// TIA Portal V17 export
// export: Created 2023-09-10T16:27:48.4257814Z, ExportSetting WithDefaults, DisplayName Totally Integrated Automation Portal, DisplayVersion V17, DisplayName TIA Portal Openness, DisplayVersion V17, DisplayName TIA Portal Version Control Interface, DisplayVersion V17, DisplayName STEP 7 Professional, DisplayVersion V17, DisplayName STEP 7 Safety, DisplayVersion V17, DisplayName WinCC Advanced, DisplayVersion V17
ORGANIZATION_BLOCK "Main"   // OB1, LAD, ProgramCycle
TITLE = "Main Program Sweep (Cycle)"
{ S7_Optimized_Access := 'TRUE' }
VERSION : 0.1
// stored: AutoNumber true, IsIECCheckEnabled false, SetENOAutomatically false
   VAR_INPUT
      Initial_Call : Bool;   // Initial call of this OB
      Remanence : Bool;   // =True, if remanent data are available
   END_VAR
   VAR_TEMP
      turn : Int;
      machinePosition : DInt;
   END_VAR
   VAR_TEMP   // added for the SCL form of the ladder/FBD networks
      _w1 : Bool;
      _w2 : Bool;
      _w3 : Bool;
   END_VAR
BEGIN

REGION Network 1: Encoder modbus function
   // te
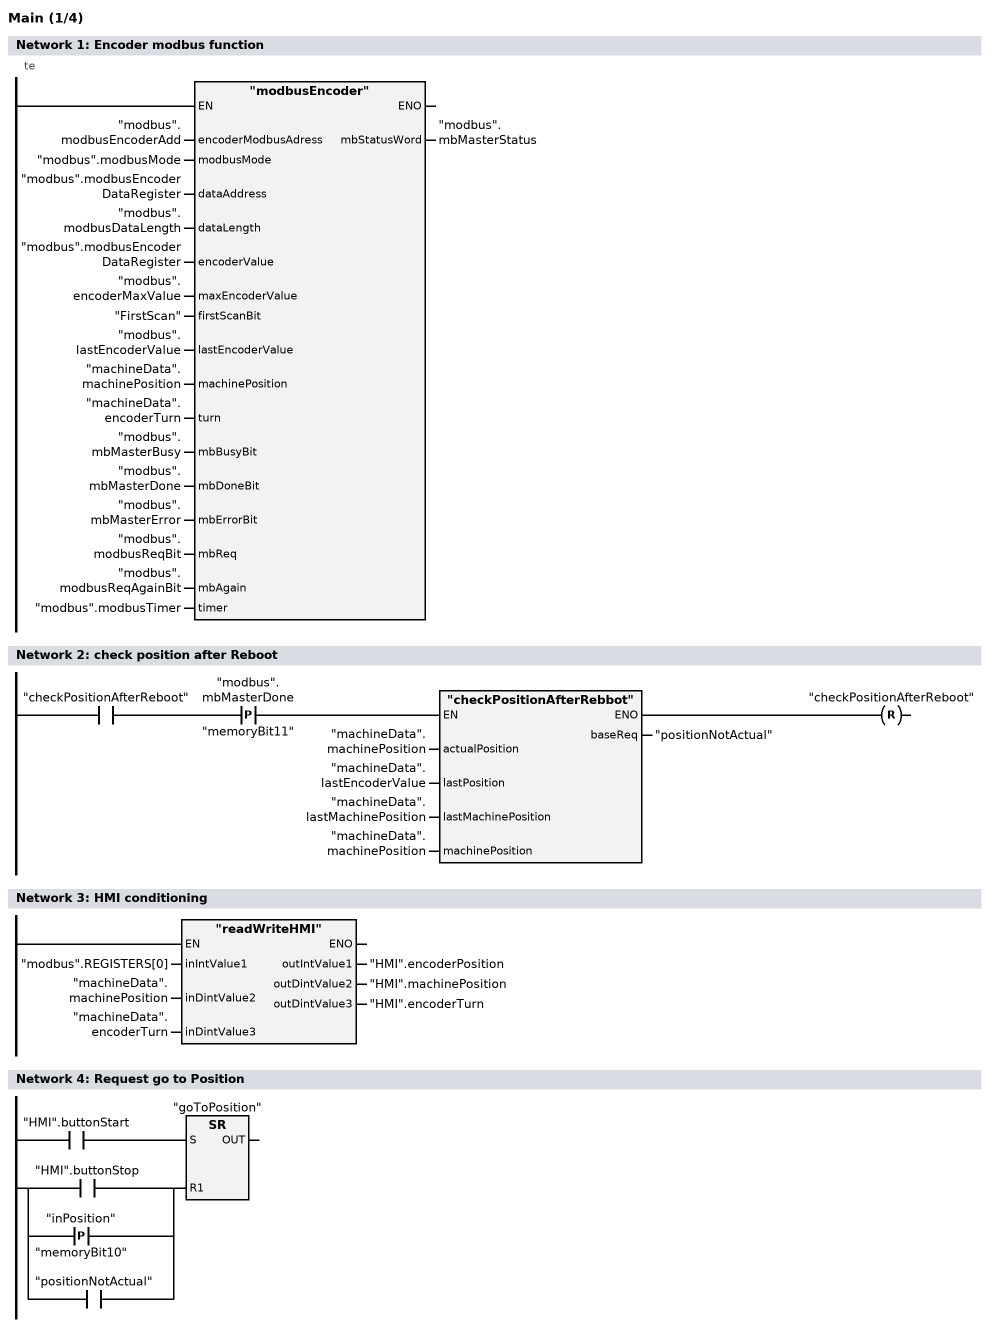
   RUNG wire#powerrail
      "modbusEncoder"(encoderModbusAdress := "modbus".modbusEncoderAdd, modbusMode := "modbus".modbusMode, dataAddress := "modbus".modbusEncoderDataRegister, dataLength := "modbus".modbusDataLength, encoderValue := "modbus".modbusEncoderDataRegister, maxEncoderValue := "modbus".encoderMaxValue, firstScanBit := "FirstScan", lastEncoderValue := "modbus".lastEncoderValue, machinePosition := "machineData".machinePosition, turn := "machineData".encoderTurn, mbBusyBit := "modbus".mbMasterBusy, mbDoneBit := "modbus".mbMasterDone, mbErrorBit := "modbus".mbMasterError, mbReq := "modbus".modbusReqBit, mbAgain := "modbus".modbusReqAgainBit, "timer" := "modbus".modbusTimer, mbStatusWord => "modbus".mbMasterStatus)
   END_RUNG
   // the same network as SCL:
   "modbusEncoder"(encoderModbusAdress := "modbus".modbusEncoderAdd,
                   modbusMode := "modbus".modbusMode,
                   dataAddress := "modbus".modbusEncoderDataRegister,
                   dataLength := "modbus".modbusDataLength,
                   encoderValue := "modbus".modbusEncoderDataRegister,
                   maxEncoderValue := "modbus".encoderMaxValue,
                   firstScanBit := "FirstScan",
                   lastEncoderValue := "modbus".lastEncoderValue,
                   machinePosition := "machineData".machinePosition,
                   turn := "machineData".encoderTurn,
                   mbBusyBit := "modbus".mbMasterBusy,
                   mbDoneBit := "modbus".mbMasterDone,
                   mbErrorBit := "modbus".mbMasterError,
                   mbReq := "modbus".modbusReqBit,
                   mbAgain := "modbus".modbusReqAgainBit,
                   "timer" := "modbus".modbusTimer,
                   mbStatusWord => "modbus".mbMasterStatus);
END_REGION

REGION Network 2: check position after Reboot
   RUNG wire#powerrail
      Contact( "checkPositionAfterReboot" )
      P_Contact(operand := "modbus".mbMasterDone, bit := "memoryBit11")
      "checkPositionAfterRebbot"(actualPosition := "machineData".machinePosition, lastPosition := "machineData".lastEncoderValue, lastMachinePosition := "machineData".lastMachinePosition, machinePosition := "machineData".machinePosition, baseReq => "positionNotActual")
      R_Coil( "checkPositionAfterReboot" )
   END_RUNG
   // the same network as SCL:
   #_w1 := "checkPositionAfterReboot" AND "modbus".mbMasterDone AND NOT "memoryBit11";   // rising edge of "modbus".mbMasterDone
   "memoryBit11" := "modbus".mbMasterDone;
   "checkPositionAfterRebbot"(EN := #_w1,
                           actualPosition := "machineData".machinePosition,
                           lastPosition := "machineData".lastEncoderValue,
                           lastMachinePosition := "machineData".lastMachinePosition,
                           machinePosition := "machineData".machinePosition,
                           baseReq => "positionNotActual",
                           ENO => #_w2);
   IF #_w2 THEN "checkPositionAfterReboot" := FALSE; END_IF;
END_REGION

REGION Network 3: HMI conditioning
   RUNG wire#powerrail
      "readWriteHMI"(inIntValue1 := "modbus".REGISTERS[0], inDintValue2 := "machineData".machinePosition, inDintValue3 := "machineData".encoderTurn, outIntValue1 => "HMI".encoderPosition, outDintValue2 => "HMI".machinePosition, outDintValue3 => "HMI".encoderTurn)
   END_RUNG
   // the same network as SCL:
   "readWriteHMI"(inIntValue1 := "modbus".REGISTERS[0],
                  inDintValue2 := "machineData".machinePosition,
                  inDintValue3 := "machineData".encoderTurn,
                  outIntValue1 => "HMI".encoderPosition,
                  outDintValue2 => "HMI".machinePosition,
                  outDintValue3 => "HMI".encoderTurn);
END_REGION

REGION Network 4: Request go to Position
   RUNG wire#powerrail
      Contact( "HMI".buttonStart )
      S_SR(operand := "goToPosition", r1 := wire#w1)
   END_RUNG
   RUNG wire#powerrail
      Contact( "HMI".buttonStop )
   END_RUNG wire#w1
   RUNG wire#powerrail
      P_Contact(operand := "inPosition", bit := "memoryBit10")
   END_RUNG wire#w1
   RUNG wire#powerrail
      Contact( "positionNotActual" )
   END_RUNG wire#w1
   // the same network as SCL:
   #_w1 := "inPosition" AND NOT "memoryBit10";   // rising edge of "inPosition"
   "memoryBit10" := "inPosition";
   IF "HMI".buttonStart THEN
       "goToPosition" := TRUE;   // SR flip-flop
   END_IF;
   IF "HMI".buttonStop OR #_w1 OR "positionNotActual" THEN "goToPosition" := FALSE; END_IF;
END_REGION

REGION Network 5: Homing
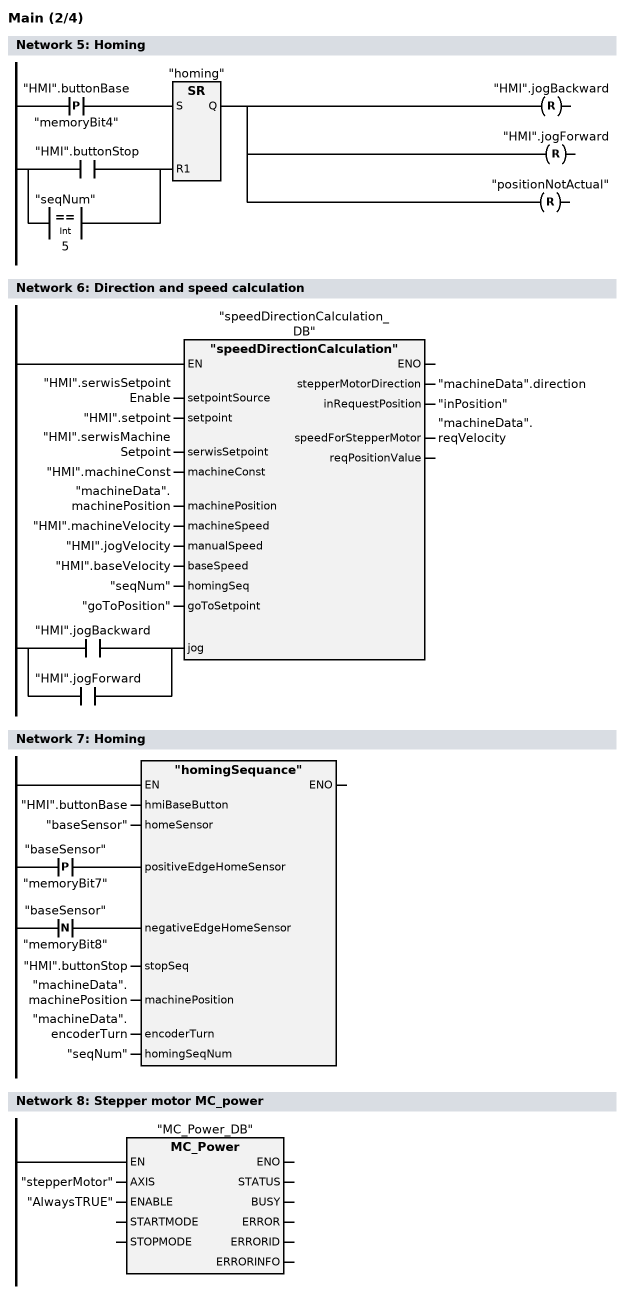
   RUNG wire#powerrail
      P_Contact(operand := "HMI".buttonBase, bit := "memoryBit4")
      S_SR(operand := "homing", r1 := wire#w1)
      wire#w2
      R_Coil( "HMI".jogBackward )
   END_RUNG
   RUNG wire#powerrail
      Contact( "HMI".buttonStop )
   END_RUNG wire#w1
   RUNG wire#powerrail
      { S7_Templates := "SrcType := Int" } EQ_Contact(in1 := "seqNum", in2 := 5)
   END_RUNG wire#w1
   RUNG wire#w2
      R_Coil( "HMI".jogForward )
   END_RUNG
   RUNG wire#w2
      R_Coil( "positionNotActual" )
   END_RUNG
   // the same network as SCL:
   #_w1 := "HMI".buttonBase AND NOT "memoryBit4";   // rising edge of "HMI".buttonBase
   "memoryBit4" := "HMI".buttonBase;
   IF #_w1 THEN
       "homing" := TRUE;   // SR flip-flop
   END_IF;
   IF "HMI".buttonStop OR ("seqNum" = 5) THEN "homing" := FALSE; END_IF;
   IF "homing" THEN
       "HMI".jogBackward := FALSE;
       "HMI".jogForward := FALSE;
       "positionNotActual" := FALSE;
   END_IF;
END_REGION

REGION Network 6: Direction and speed calculation
   RUNG wire#powerrail
      "speedDirectionCalculation_DB"(jog := wire#w1, setpointSource := "HMI".serwisSetpointEnable, setpoint := "HMI".setpoint, serwisSetpoint := "HMI".serwisMachineSetpoint, machineConst := "HMI".machineConst, machinePosition := "machineData".machinePosition, machineSpeed := "HMI".machineVelocity, manualSpeed := "HMI".jogVelocity, baseSpeed := "HMI".baseVelocity, homingSeq := "seqNum", goToSetpoint := "goToPosition", stepperMotorDirection => "machineData".direction, inRequestPosition => "inPosition", speedForStepperMotor => "machineData".reqVelocity, reqPositionValue =>)
   END_RUNG
   RUNG wire#powerrail
      Contact( "HMI".jogBackward )
   END_RUNG wire#w1
   RUNG wire#powerrail
      Contact( "HMI".jogForward )
   END_RUNG wire#w1
   // the same network as SCL:
   "speedDirectionCalculation_DB"(setpointSource := "HMI".serwisSetpointEnable,   // "speedDirectionCalculation"
                           setpoint := "HMI".setpoint,
                           serwisSetpoint := "HMI".serwisMachineSetpoint,
                           machineConst := "HMI".machineConst,
                           machinePosition := "machineData".machinePosition,
                           machineSpeed := "HMI".machineVelocity,
                           manualSpeed := "HMI".jogVelocity,
                           baseSpeed := "HMI".baseVelocity,
                           homingSeq := "seqNum",
                           goToSetpoint := "goToPosition",
                           jog := "HMI".jogBackward OR "HMI".jogForward,
                           stepperMotorDirection => "machineData".direction,
                           inRequestPosition => "inPosition",
                           speedForStepperMotor => "machineData".reqVelocity);
END_REGION

REGION Network 7: Homing
   RUNG wire#powerrail
      "homingSequance"(positiveEdgeHomeSensor := wire#w1, negativeEdgeHomeSensor := wire#w2, hmiBaseButton := "HMI".buttonBase, homeSensor := "baseSensor", stopSeq := "HMI".buttonStop, machinePosition := "machineData".machinePosition, encoderTurn := "machineData".encoderTurn, homingSeqNum := "seqNum")
   END_RUNG
   RUNG wire#powerrail
      P_Contact(operand := "baseSensor", bit := "memoryBit7")
   END_RUNG wire#w1
   RUNG wire#powerrail
      N_Contact(operand := "baseSensor", bit := "memoryBit8")
   END_RUNG wire#w2
   // the same network as SCL:
   #_w1 := "baseSensor" AND NOT "memoryBit7";   // rising edge of "baseSensor"
   "memoryBit7" := "baseSensor";
   #_w2 := NOT "baseSensor" AND "memoryBit8";   // falling edge of "baseSensor"
   "memoryBit8" := "baseSensor";
   "homingSequance"(hmiBaseButton := "HMI".buttonBase,
                    homeSensor := "baseSensor",
                    positiveEdgeHomeSensor := #_w1,
                    negativeEdgeHomeSensor := #_w2,
                    stopSeq := "HMI".buttonStop,
                    machinePosition := "machineData".machinePosition,
                    encoderTurn := "machineData".encoderTurn,
                    homingSeqNum := "seqNum");
END_REGION

REGION Network 8: Stepper motor MC_power
   RUNG wire#powerrail
      "MC_Power_DB".MC_Power(Axis := "stepperMotor", Enable := "AlwaysTRUE", StartMode :=, StopMode :=, Status =>, Busy =>, Error =>, ErrorID =>, ErrorInfo =>)
   END_RUNG
   // the same network as SCL:
   "MC_Power_DB"(Axis := "stepperMotor", Enable := "AlwaysTRUE");   // MC_Power
END_REGION

REGION Network 9: Srepper motor drive
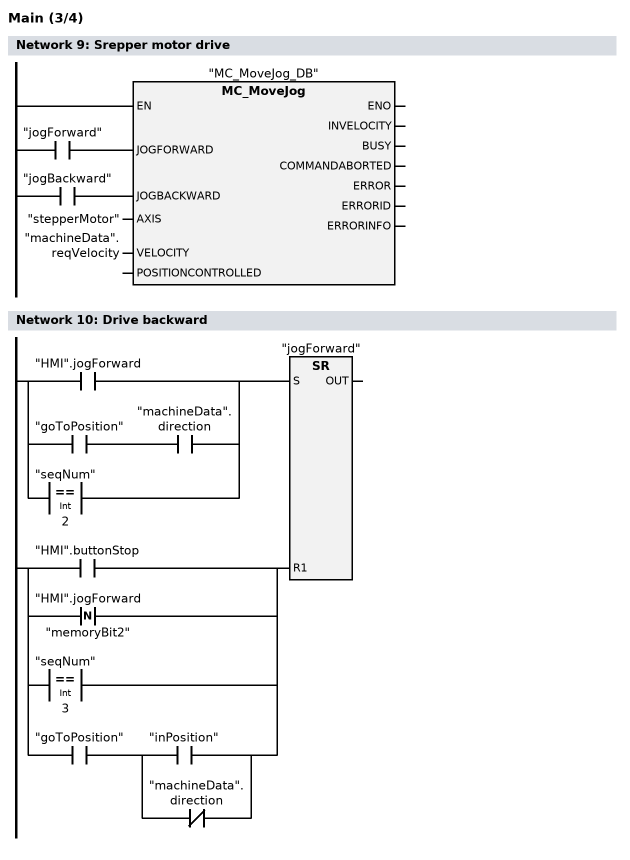
   RUNG wire#powerrail
      "MC_MoveJog_DB".MC_MoveJog(JogForward := wire#w1, JogBackward := wire#w2, Axis := "stepperMotor", Velocity := "machineData".reqVelocity, PositionControlled :=, InVelocity =>, Busy =>, CommandAborted =>, Error =>, ErrorID =>, ErrorInfo =>)
   END_RUNG
   RUNG wire#powerrail
      Contact( "jogForward" )
   END_RUNG wire#w1
   RUNG wire#powerrail
      Contact( "jogBackward" )
   END_RUNG wire#w2
   // the same network as SCL:
   "MC_MoveJog_DB"(JogForward := "jogForward",   // MC_MoveJog
                   JogBackward := "jogBackward",
                   Axis := "stepperMotor",
                   Velocity := "machineData".reqVelocity);
END_REGION

REGION Network 10: Drive backward
   RUNG wire#powerrail
      Contact( "HMI".jogForward )
      wire#w1
      S_SR(operand := "jogForward", r1 := wire#w3)
   END_RUNG
   RUNG wire#powerrail
      Contact( "goToPosition" )
      Contact( "machineData".direction )
   END_RUNG wire#w1
   RUNG wire#powerrail
      { S7_Templates := "SrcType := Int" } EQ_Contact(in1 := "seqNum", in2 := 2)
   END_RUNG wire#w1
   RUNG wire#powerrail
      Contact( "HMI".buttonStop )
   END_RUNG wire#w3
   RUNG wire#powerrail
      N_Contact(operand := "HMI".jogForward, bit := "memoryBit2")
   END_RUNG wire#w3
   RUNG wire#powerrail
      { S7_Templates := "SrcType := Int" } EQ_Contact(in1 := "seqNum", in2 := 3)
   END_RUNG wire#w3
   RUNG wire#powerrail
      Contact( "goToPosition" )
      wire#w2
      Contact( "inPosition" )
   END_RUNG wire#w3
   RUNG wire#w2
      I_Contact( "machineData".direction )
   END_RUNG wire#w3
   // the same network as SCL:
   #_w1 := NOT "HMI".jogForward AND "memoryBit2";   // falling edge of "HMI".jogForward
   "memoryBit2" := "HMI".jogForward;
   IF "HMI".jogForward OR ("goToPosition" AND "machineData".direction) OR ("seqNum" = 2) THEN
       "jogForward" := TRUE;   // SR flip-flop
   END_IF;
   IF "HMI".buttonStop OR #_w1 OR ("seqNum" = 3) OR ("goToPosition" AND ("inPosition" OR NOT "machineData".direction)) THEN
       "jogForward" := FALSE;
   END_IF;
END_REGION

REGION Network 11: Drive forward
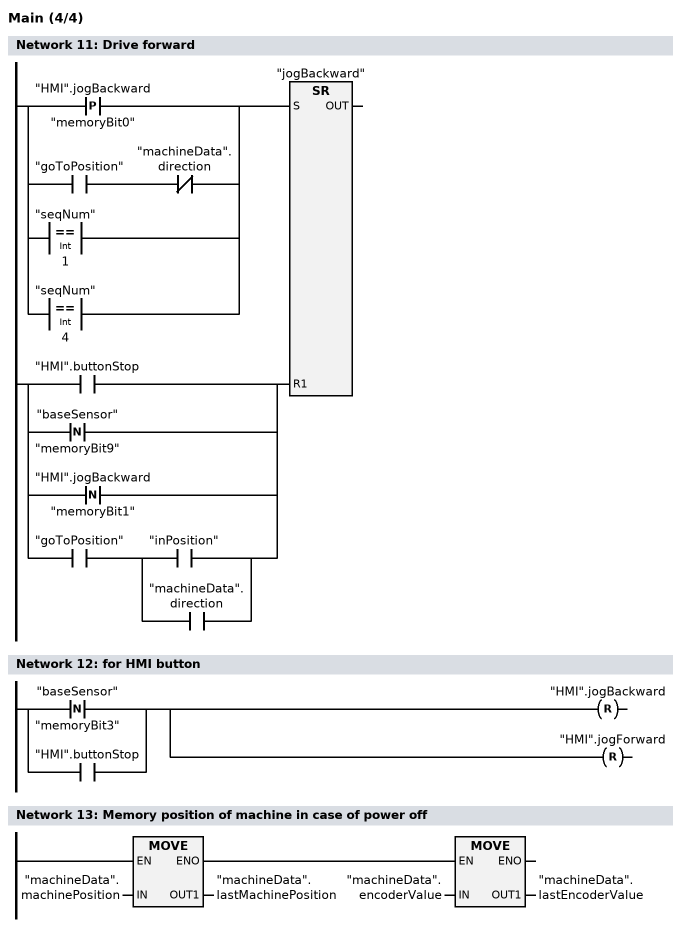
   RUNG wire#powerrail
      P_Contact(operand := "HMI".jogBackward, bit := "memoryBit0")
      wire#w1
      S_SR(operand := "jogBackward", r1 := wire#w3)
   END_RUNG
   RUNG wire#powerrail
      Contact( "goToPosition" )
      I_Contact( "machineData".direction )
   END_RUNG wire#w1
   RUNG wire#powerrail
      { S7_Templates := "SrcType := Int" } EQ_Contact(in1 := "seqNum", in2 := 1)
   END_RUNG wire#w1
   RUNG wire#powerrail
      { S7_Templates := "SrcType := Int" } EQ_Contact(in1 := "seqNum", in2 := 4)
   END_RUNG wire#w1
   RUNG wire#powerrail
      Contact( "HMI".buttonStop )
   END_RUNG wire#w3
   RUNG wire#powerrail
      N_Contact(operand := "baseSensor", bit := "memoryBit9")
   END_RUNG wire#w3
   RUNG wire#powerrail
      N_Contact(operand := "HMI".jogBackward, bit := "memoryBit1")
   END_RUNG wire#w3
   RUNG wire#powerrail
      Contact( "goToPosition" )
      wire#w2
      Contact( "inPosition" )
   END_RUNG wire#w3
   RUNG wire#w2
      Contact( "machineData".direction )
   END_RUNG wire#w3
   // the same network as SCL:
   #_w1 := "HMI".jogBackward AND NOT "memoryBit0";   // rising edge of "HMI".jogBackward
   "memoryBit0" := "HMI".jogBackward;
   #_w2 := NOT "baseSensor" AND "memoryBit9";   // falling edge of "baseSensor"
   "memoryBit9" := "baseSensor";
   #_w3 := NOT "HMI".jogBackward AND "memoryBit1";   // falling edge of "HMI".jogBackward
   "memoryBit1" := "HMI".jogBackward;
   IF #_w1 OR ("goToPosition" AND NOT "machineData".direction) OR ("seqNum" = 1) OR ("seqNum" = 4) THEN
       "jogBackward" := TRUE;   // SR flip-flop
   END_IF;
   IF "HMI".buttonStop OR #_w2 OR #_w3 OR ("goToPosition" AND ("inPosition" OR "machineData".direction)) THEN
       "jogBackward" := FALSE;
   END_IF;
END_REGION

REGION Network 12: for HMI button
   RUNG wire#powerrail
      N_Contact(operand := "baseSensor", bit := "memoryBit3")
      wire#w1
      R_Coil( "HMI".jogBackward )
   END_RUNG
   RUNG wire#powerrail
      Contact( "HMI".buttonStop )
   END_RUNG wire#w1
   RUNG wire#w1
      R_Coil( "HMI".jogForward )
   END_RUNG
   // the same network as SCL:
   #_w1 := NOT "baseSensor" AND "memoryBit3";   // falling edge of "baseSensor"
   "memoryBit3" := "baseSensor";
   IF #_w1 OR "HMI".buttonStop THEN
       "HMI".jogBackward := FALSE;
       "HMI".jogForward := FALSE;
   END_IF;
END_REGION

REGION Network 13: Memory position of machine in case of power off
   RUNG wire#powerrail
      Move(in := "machineData".machinePosition, out1 => "machineData".lastMachinePosition)
      Move(in := "machineData".encoderValue, out1 => "machineData".lastEncoderValue)
   END_RUNG
   // the same network as SCL:
   "machineData".lastMachinePosition := "machineData".machinePosition;
   "machineData".lastEncoderValue := "machineData".encoderValue;
END_REGION
END_ORGANIZATION_BLOCK
